TYPE MeasurementConfig :
STRUCT
	///Is the quantity being measured? (Can be false e.g. if the sensor is deliberately not connected (yet).)
	enabled: BOOL;
	///Offset to be added to the measured value (default: 0 = no offset)
	offset: LREAL;
	///Config
	alarms: HiHiLoLoAlarmConfig;
END_STRUCT
END_TYPE

(* stored: Version 1.1.0.1, ProductVersion 3.1.4019.2
   DUT MeasurementConfig: Id {35667af7-a410-4d51-b349-1c5d8309cbde} *)
